INTERFACE I_MotionAxisCommon

PROPERTY AxisState : MC_AxisStates
GET
END_GET
END_PROPERTY

PROPERTY BufferMode : MC_BufferMode
SET
END_SET
END_PROPERTY

PROPERTY Busy : BOOL
GET
END_GET
END_PROPERTY

PROPERTY Cmd : UINT
SET
END_SET
END_PROPERTY

PROPERTY CmdData : UINT
SET
END_SET
END_PROPERTY

PROPERTY CmdHalt : BOOL
GET
END_GET
SET
END_SET
END_PROPERTY

PROPERTY CmdMoveAbsolute : BOOL
GET
END_GET
SET
END_SET
END_PROPERTY

PROPERTY CmdMoveHome : BOOL
GET
END_GET
SET
END_SET
END_PROPERTY

PROPERTY CmdReset : BOOL
GET
END_GET
SET
END_SET
END_PROPERTY

PROPERTY Command : UINT
SET
END_SET
END_PROPERTY

PROPERTY CommandAborted : BOOL
GET
END_GET
END_PROPERTY

PROPERTY CommandData : UINT
SET
END_SET
END_PROPERTY

PROPERTY CommandedHalt : BOOL
GET
END_GET
SET
END_SET
END_PROPERTY

PROPERTY CommandedMoveAbsolute : BOOL
GET
END_GET
SET
END_SET
END_PROPERTY

PROPERTY CommandedReset : BOOL
GET
END_GET
SET
END_SET
END_PROPERTY

PROPERTY Done : BOOL
GET
END_GET
END_PROPERTY

PROPERTY EncoderCount : UDINT
GET
END_GET
END_PROPERTY

PROPERTY Error : BOOL
GET
END_GET
END_PROPERTY

PROPERTY ErrorID : UDINT
GET
END_GET
END_PROPERTY

PROPERTY ErrorMessage : STRING
GET
END_GET
END_PROPERTY

PROPERTY ExecHome : BOOL
GET
END_GET
SET
END_SET
END_PROPERTY

PROPERTY ExecMove : BOOL
GET
END_GET
SET
END_SET
END_PROPERTY

PROPERTY HaltBusy : BOOL
GET
END_GET
END_PROPERTY

PROPERTY HaltDone : BOOL
GET
END_GET
END_PROPERTY

PROPERTY HaltErrorID : UDINT
GET
END_GET
END_PROPERTY

PROPERTY HomeBusy : BOOL
GET
END_GET
END_PROPERTY

PROPERTY HomeDone : BOOL
GET
END_GET
END_PROPERTY

PROPERTY HomeError : BOOL
GET
END_GET
END_PROPERTY

PROPERTY HomeErrorID : UDINT
GET
END_GET
END_PROPERTY

PROPERTY HomeInterrupted : BOOL
GET
END_GET
END_PROPERTY

PROPERTY HomeMode : E_EpicsHomeCmd
GET
END_GET
SET
END_SET
END_PROPERTY

PROPERTY HomePosition : LREAL
GET
END_GET
SET
END_SET
END_PROPERTY

PROPERTY InTargetPosition : BOOL
GET
END_GET
END_PROPERTY

PROPERTY Interrupted : BOOL
GET
END_GET
END_PROPERTY

METHOD InterruptMove
VAR_INPUT
END_VAR
END_METHOD

PROPERTY MeasuredAcceleration : LREAL
GET
END_GET
END_PROPERTY

PROPERTY MeasuredPosition : LREAL
GET
END_GET
END_PROPERTY

PROPERTY MeasuredPositionDiff : LREAL
GET
END_GET
END_PROPERTY

PROPERTY MeasuredVelocity : LREAL
GET
END_GET
END_PROPERTY

PROPERTY ModeOfOperation : SINT
GET
END_GET
SET
END_SET
END_PROPERTY

PROPERTY MoveAbsoluteBusy : BOOL
GET
END_GET
END_PROPERTY

PROPERTY MoveAbsoluteDone : BOOL
GET
END_GET
END_PROPERTY

PROPERTY MoveAbsoluteError : BOOL
GET
END_GET
END_PROPERTY

PROPERTY MoveAbsoluteErrorID : UDINT
GET
END_GET
END_PROPERTY

PROPERTY MoveAbsoluteTargetAcceleration : LREAL
GET
END_GET
SET
END_SET
END_PROPERTY

PROPERTY MoveAbsoluteTargetDeceleration : LREAL
GET
END_GET
SET
END_SET
END_PROPERTY

PROPERTY MoveAbsoluteTargetJerk : LREAL
GET
END_GET
SET
END_SET
END_PROPERTY

PROPERTY MoveAbsoluteTargetPosition : LREAL
GET
END_GET
SET
END_SET
END_PROPERTY

PROPERTY MoveAbsoluteTargetVelocity : LREAL
GET
END_GET
SET
END_SET
END_PROPERTY

PROPERTY MoveMode : E_MoveMode
GET
END_GET
SET
END_SET
END_PROPERTY

PROPERTY Name : STRING
GET
END_GET
SET
END_SET
END_PROPERTY

PROPERTY NCParamsReadInit : BOOL
GET
END_GET
END_PROPERTY

PROPERTY NegativeMotionIsEnabled : BOOL
GET
END_GET
END_PROPERTY

PROPERTY PositiveMotionIsEnabled : BOOL
GET
END_GET
END_PROPERTY

PROPERTY PowerEnable : BOOL
GET
END_GET
SET
END_SET
END_PROPERTY

PROPERTY PowerEnableNegative : BOOL
GET
END_GET
SET
END_SET
END_PROPERTY

PROPERTY PowerEnablePositive : BOOL
GET
END_GET
SET
END_SET
END_PROPERTY

PROPERTY PowerError : BOOL
GET
END_GET
END_PROPERTY

PROPERTY PowerErrorID : UDINT
GET
END_GET
END_PROPERTY

PROPERTY PowerIsEnabled : BOOL
GET
END_GET
END_PROPERTY

PROPERTY PowerOverride : LREAL
GET
END_GET
SET
END_SET
END_PROPERTY

PROPERTY PowerStatus : BOOL
GET
END_GET
END_PROPERTY

PROPERTY RefreshDelay : TIME
GET
END_GET
SET
END_SET
END_PROPERTY

PROPERTY RefVeloSearch : LREAL
GET
END_GET
END_PROPERTY

PROPERTY RefVeloSync : LREAL
GET
END_GET
END_PROPERTY

PROPERTY ResetBusy : BOOL
GET
END_GET
END_PROPERTY

PROPERTY ResetDone : BOOL
GET
END_GET
END_PROPERTY

PROPERTY ResetError : BOOL
GET
END_GET
END_PROPERTY

PROPERTY ResetErrorID : UDINT
GET
END_GET
END_PROPERTY

PROPERTY RestoreDone : BOOL
GET
END_GET
SET
END_SET
END_PROPERTY

PROPERTY RestoreError : BOOL
GET
END_GET
END_PROPERTY

PROPERTY RestoreErrorID : UDINT
GET
END_GET
END_PROPERTY

PROPERTY SavedPosition : LREAL
GET
END_GET
END_PROPERTY

PROPERTY Servo : BOOL
GET
END_GET
SET
END_SET
END_PROPERTY

(* 
	Check all post condition before updating bCommandedMoveAbsolute
	The implmentatation will depend on the axis type
	DS402 NC/Direct axis : Implementation need to check that the drive is in the correct mode before initaiting the move then set bCommandedMoveAbsolute
	MP NC axis : will immediately write to bCommandedMoveAbsolute 
*)
METHOD StartMove : BOOL
VAR_INPUT
END_VAR
END_METHOD

METHOD StopMove
VAR_INPUT
END_VAR
END_METHOD

END_INTERFACE

(* stored: Version 1.1.0.1
   Itf I_MotionAxisCommon: Id {df11a94c-15fb-4aec-9011-b2ef3c6b1fb4}
   Property AxisState: Id {fbced42b-bd0e-4f8b-9d53-090d7101c00b}
   Get Get: Id {3f69a59a-8937-4e06-aeb3-542997f1671d}
   Property BufferMode: Id {38f05b0c-8759-4cb0-852d-594c9ce9b628}
   Set Set: Id {b31efd89-9be0-445c-8e9c-f516f7340490}
   Property Busy: Id {1dc67c19-7944-41b9-ba51-efc9922261f1}
   Get Get: Id {a5860cad-3e89-42b7-8b83-9419c9d09efd}
   Property Cmd: Id {69b39c97-9b90-4d9b-a9e7-485ac83933e1}
   Set Set: Id {abefe843-77e6-4997-be3a-c32a08ca8c8f}
   Property CmdData: Id {054016e0-1db6-4015-9b60-d4eac71effd1}
   Set Set: Id {fc9b83c4-f2f9-46c4-bd97-0ba0143c91d4}
   Property CmdHalt: Id {c0746e6c-e503-4768-b680-1d04f0ae1984}
   Get Get: Id {6a9152b5-e347-4fca-96b2-7284ad169bbc}
   Set Set: Id {98676a7a-0323-4266-9c73-239c40deb92e}
   Property CmdMoveAbsolute: Id {f4037a53-e108-4ca0-9a92-314a66e74287}
   Get Get: Id {447a2d74-14ca-4065-b818-42aaec9a8873}
   Set Set: Id {2137edf8-e503-4512-a064-4f3f78293549}
   Property CmdMoveHome: Id {c447ca24-e237-4885-a9a3-281864c8338b}
   Get Get: Id {bd009231-61d7-4bed-ae68-5c589c9f60c3}
   Set Set: Id {fd07a648-391b-4835-a127-b5f46d9080b8}
   Property CmdReset: Id {d517a452-024b-4976-921a-8fe69a2bf16f}
   Get Get: Id {50257a3a-da8e-4338-964f-dc07fa89e7aa}
   Set Set: Id {056030c6-8ce9-46ea-b6e0-3abbc748c572}
   Property Command: Id {7b9a7e1c-dedf-411f-ad91-f5efd6c329ee}
   Set Set: Id {c20cbc5e-5c11-4ee7-af97-18507def7d36}
   Property CommandAborted: Id {0fa2c2c2-ee04-43d1-b494-0f4602cb897b}
   Get Get: Id {b918462e-6014-4e11-9e53-215e9c34e70a}
   Property CommandData: Id {0e8b4985-8f01-4f1b-8087-81dc02998277}
   Set Set: Id {e5aa3541-32bf-49db-9fad-772fe065c88c}
   Property CommandedHalt: Id {28caa621-b1b5-45c3-948b-355529ae63c2}
   Get Get: Id {9fc451d3-9985-4a65-a079-615be98f9e47}
   Set Set: Id {afbd26a2-5d4f-4673-a5ff-92792f920642}
   Property CommandedMoveAbsolute: Id {be1022ab-c175-45cf-b747-4904f7dbb61a}
   Get Get: Id {2b465d88-c80e-452d-bd64-a4daa37a937f}
   Set Set: Id {148eb03e-69c6-4884-b363-b91c6e29515e}
   Property CommandedReset: Id {cd7e8bfd-a0cf-4671-a69b-1557a160bd00}
   Get Get: Id {cc6afb54-414e-4354-b571-2acc42bfca27}
   Set Set: Id {367e203b-5f9b-41d7-9061-a806fa5317d7}
   Property Done: Id {7ff11c7c-614b-47cb-baec-d0e1b99b56ef}
   Get Get: Id {731f59b1-4ebc-46a2-8ec3-b8482a33696e}
   Property EncoderCount: Id {9e7da4f2-c20f-41ff-89bb-b6a6d51aa2c8}
   Get Get: Id {e6419d2f-35cd-4088-84a8-5db9b615087b}
   Property Error: Id {1839383d-e5fd-4221-a255-d379f863c6e8}
   Get Get: Id {3b6a6767-2e6d-4d83-ac0a-858e93b4acb4}
   Property ErrorID: Id {a8ca6773-3b68-40ff-aa9d-b90cfd491bbf}
   Get Get: Id {3c8f7f0c-cdf8-46a2-b2ed-eae80213300d}
   Property ErrorMessage: Id {62e7f2d7-0787-4e90-bcb4-6a79cccb37fe}
   Get Get: Id {540b8f36-640c-487f-bfb4-5e6df636128d}
   Property ExecHome: Id {6e6bf230-720c-4613-80af-c8c009118fd1}
   Get Get: Id {6125f9cc-b415-4a4e-b052-4c188af3488f}
   Set Set: Id {7f9e6770-dd66-4322-8ad8-27eaa7f2abde}
   Property ExecMove: Id {9fe3d498-d752-48dc-aa3d-5d4c1306ffed}
   Get Get: Id {a97d3154-60d9-4bed-b64b-6f7f0fa20999}
   Set Set: Id {df2886f7-a831-4b24-b707-10da4aeec211}
   Property HaltBusy: Id {5eefa523-d59e-4ef7-b5af-021b09543db4}
   Get Get: Id {e59b7e42-9140-4829-bc23-b10577952d4c}
   Property HaltDone: Id {2708b684-0763-4c58-ad74-2f54f4c3351c}
   Get Get: Id {1696e0d8-0e21-4edb-aa6d-6c70bfdba3fc}
   Property HaltErrorID: Id {76c342d8-ef7a-4cbf-b33e-fe9701803b90}
   Get Get: Id {84f9ea8e-6e1e-480a-86db-80a8046724f4}
   Property HomeBusy: Id {d6d79540-89df-4e37-8d40-761027f4650a}
   Get Get: Id {2085b480-133e-431e-af2b-2e28067f5fcf}
   Property HomeDone: Id {6d82612d-3be0-411d-9fbb-4db9d5b30e7a}
   Get Get: Id {dc264365-5ed4-4cc8-8938-a641a37a624b}
   Property HomeError: Id {66345dd5-8f9b-4c6e-862e-018015cab45f}
   Get Get: Id {bf4a9cda-c749-44e3-b222-0aa2dcfcebdb}
   Property HomeErrorID: Id {5637a821-11d4-4cf6-b60b-88d54de78092}
   Get Get: Id {522d3d81-d3e7-4960-90e6-f89bf9e2f7eb}
   Property HomeInterrupted: Id {e35df6e5-941d-4778-a7be-e76d3f381d59}
   Get Get: Id {58767f79-ed58-4276-8041-a41052c97a6b}
   Property HomeMode: Id {32879e99-b015-407a-b611-ffd5ee8ac39d}
   Get Get: Id {16a9aefe-77f3-400a-84d1-c01ba499762b}
   Set Set: Id {7d19f097-4494-4927-be4b-078feb862d60}
   Property HomePosition: Id {292c1204-dc74-485b-8911-177c01a78ff8}
   Get Get: Id {9ffd7eeb-12d8-4c9d-8056-57cabd96be13}
   Set Set: Id {3692be77-4178-4aa1-b1e2-16325bc48cb0}
   Property InTargetPosition: Id {79a34037-a39e-4bee-ab9e-d3c72c400a3c}
   Get Get: Id {c1b81aa3-9460-4489-85a7-c42e28336f83}
   Property Interrupted: Id {498fa652-b5b3-4e1f-976d-8ce99932c93a}
   Get Get: Id {2c6824d4-b3f4-460d-9f3f-bc04fc1c06c7}
   Method InterruptMove: Id {303223bb-9993-4d05-b3de-df5e0ce6e8a3}
   Property MeasuredAcceleration: Id {d4d9e574-a194-4fa2-98b9-07d056a1260a}
   Get Get: Id {64393f7d-024e-4f33-8143-f1be9ffe5b8f}
   Property MeasuredPosition: Id {d63c1cdc-d7a8-436e-8781-271d2fcb7da2}
   Get Get: Id {36e1d037-35d3-410b-bb6f-e4f6e0d800dc}
   Property MeasuredPositionDiff: Id {4962ee10-def8-4f9d-bf3b-0b44ac0ece59}
   Get Get: Id {fc230d1f-c943-4ec1-a46d-a7979d2b7069}
   Property MeasuredVelocity: Id {ba169ffc-f0a6-4913-8469-66deff516709}
   Get Get: Id {62daf172-9d22-4bb4-bfac-abdfd22e6c7b}
   Property ModeOfOperation: Id {e6ef5f87-d9f5-4819-a545-2bdc671caace}
   Get Get: Id {5767ff6c-d328-42fc-a0a0-bd49b1295ca0}
   Set Set: Id {c3f1cd01-5c5f-4eb4-afce-893c68097624}
   Property MoveAbsoluteBusy: Id {f8fb30ef-d277-418f-982b-66ef86e1769d}
   Get Get: Id {11b339b5-cdec-49fb-9600-a6ec69bc6a16}
   Property MoveAbsoluteDone: Id {84978858-3bb9-4917-be38-de8a68ac208b}
   Get Get: Id {129da105-f372-4faf-add9-30e139e5f062}
   Property MoveAbsoluteError: Id {64cf4975-3274-4a57-9bc5-8610f16695ba}
   Get Get: Id {681cadf4-083a-4ae4-a53c-86cf46221723}
   Property MoveAbsoluteErrorID: Id {4fb23927-b236-4114-ae37-f615a1b8edc0}
   Get Get: Id {a023c07f-7952-4ec4-83ec-1efda5ff2614}
   Property MoveAbsoluteTargetAcceleration: Id {70a35961-bee7-4b46-b0a3-6d71eaea287d}
   Get Get: Id {9898cff6-ce1f-4fb8-8f53-4ba3d7d4fea1}
   Set Set: Id {b2459bb9-7080-49b9-ae3a-a918cd839621}
   Property MoveAbsoluteTargetDeceleration: Id {31845d61-2b46-4eb7-89e1-f67edbd56c4f}
   Get Get: Id {9a64bf3b-7a3b-4dec-a769-9b31e5a86434}
   Set Set: Id {e7ada26d-8451-438f-b463-e10f2d3a1bb8}
   Property MoveAbsoluteTargetJerk: Id {9119fca5-a884-4a17-a499-ebd775946ce3}
   Get Get: Id {1a98813c-01e8-4cb0-8272-d799fe855c2f}
   Set Set: Id {fcaf00f7-169a-4518-82c4-db7d885f20c5}
   Property MoveAbsoluteTargetPosition: Id {4c3ad4b2-e392-4b88-8a83-082f941a6830}
   Get Get: Id {8a09bba2-a387-469e-8361-0e2306956cba}
   Set Set: Id {c58fc251-226c-4365-badb-dca9ec823ab7}
   Property MoveAbsoluteTargetVelocity: Id {08e71f81-65e6-4cad-a488-7ef932c2b524}
   Get Get: Id {d4d23ccf-3369-4604-993d-56d3faa062bc}
   Set Set: Id {0be80c1e-730f-40bc-8e47-969d994de88e}
   Property MoveMode: Id {05f924a5-d3a6-4da7-ab50-fcad0580fbfb}
   Get Get: Id {4e619b19-1227-4aa9-97bd-f7e260dcc6cd}
   Set Set: Id {2987c28d-902f-4e1a-bce2-2b0a7c7390d5}
   Property Name: Id {0c6fd7a6-29c0-4c88-879f-f0f43862e70a}
   Get Get: Id {0df1c16f-fce7-44ce-a865-4fda8703479c}
   Set Set: Id {50a58ed7-b3ae-45d2-8b55-54fab7befe10}
   Property NCParamsReadInit: Id {f843168c-ca4c-4733-b6db-f83934f20ac1}
   Get Get: Id {9c60541a-3e75-4e37-92d5-dc139cd07934}
   Property NegativeMotionIsEnabled: Id {89f73a4c-6b65-4069-892b-fbfc7e7d2963}
   Get Get: Id {82333464-dc32-4ef8-bfed-612699606e4b}
   Property PositiveMotionIsEnabled: Id {52b21291-5115-4fe8-b5cd-5d002408c68b}
   Get Get: Id {1b2b33a3-a699-41d1-89bf-9eec4d0a49ca}
   Property PowerEnable: Id {8f4626d6-0f8b-4b9d-a413-29dca15842e6}
   Get Get: Id {80cde4e4-17e9-4a07-a9cc-6347ce732266}
   Set Set: Id {b3427a42-2fec-45a1-86c8-2c735642631f}
   Property PowerEnableNegative: Id {a552419c-1e47-4ba6-86f3-9cd43b6c7d4f}
   Get Get: Id {c8e9c776-921f-42c7-a895-e64aa928906d}
   Set Set: Id {2d84af61-aa81-442f-87dd-3dcea000019a}
   Property PowerEnablePositive: Id {8a310391-dab0-4dd4-84ea-7e42d91a1c1b}
   Get Get: Id {9f36b795-1fb8-4212-83b1-d67198dca149}
   Set Set: Id {ba7d2aa7-0ae3-4c74-874c-2d6ae8f7c7cf}
   Property PowerError: Id {cb1b5b40-b70d-4a67-958a-9b06cfba612b}
   Get Get: Id {ae2b0ff5-5ffb-44e3-b875-297aa814c673}
   Property PowerErrorID: Id {4aee72fa-f2a7-431e-b4b4-0b9354d8eb3f}
   Get Get: Id {a54d7cf3-a137-4078-938e-e669e7c312e2}
   Property PowerIsEnabled: Id {1be1dbac-9180-4e18-8d7d-7ac4fb3a523a}
   Get Get: Id {dae81c77-289b-440a-8b61-e8ef6a37bede}
   Property PowerOverride: Id {db8164ef-c0bf-4e70-a366-22ab4e209738}
   Get Get: Id {a17504c2-efbb-4971-b4f3-eedbd364db39}
   Set Set: Id {ff31e593-5cb0-4acb-982d-4ad437bb4265}
   Property PowerStatus: Id {ec6d63e1-de25-46f8-a4c8-a861493a5d55}
   Get Get: Id {5341a077-011d-4b04-9806-ab379cb1f954}
   Property RefreshDelay: Id {9a60c61b-0084-4420-be8f-035904aea924}
   Get Get: Id {f1806e9b-0dce-4abd-af1d-83272cb8df1e}
   Set Set: Id {24faa0ad-b9ca-4984-a659-ab17c9d097d8}
   Property RefVeloSearch: Id {06c09a70-377d-482c-a85b-e4912b1ba011}
   Get Get: Id {1e34b3e3-2a6f-40c7-b27b-eeacf2ee48da}
   Property RefVeloSync: Id {ad7860fb-e8a6-42b6-aaff-223373b4f98f}
   Get Get: Id {62cd0a9d-dc15-48af-ae9d-14d810b2fe9f}
   Property ResetBusy: Id {252e8874-c509-40df-a935-8a5f3cbe2b7a}
   Get Get: Id {1352f413-28b0-47c7-89f3-68206fd5c6bb}
   Property ResetDone: Id {d4e08fc6-eeda-4353-a1d6-7047dbfb6a8a}
   Get Get: Id {754bf460-2d23-4adc-8924-46cc6786b79b}
   Property ResetError: Id {492c4d78-fea4-491d-9af5-1a5800d3ff0f}
   Get Get: Id {9f4ff4de-0fc6-450d-a532-1e53e644e0fc}
   Property ResetErrorID: Id {7ec9a9da-2ba3-442e-8c3f-a80607933d95}
   Get Get: Id {0adcb703-0fab-4a7a-94a7-18c9597f870e}
   Property RestoreDone: Id {852d5da2-20f3-40a4-8ab0-8b0ebb2ca285}
   Get Get: Id {4f3b62f8-9947-4e8d-a9cf-f23f4d32cb01}
   Set Set: Id {11f68748-f280-450f-b307-949684cb9a43}
   Property RestoreError: Id {80815cd7-c76d-4675-bb97-e801d3dcea69}
   Get Get: Id {dbe76bd4-2085-47ed-82a9-7ce3e56236f5}
   Property RestoreErrorID: Id {14478e39-3848-4591-86df-eb5530d2d0db}
   Get Get: Id {369bf874-f43c-4d30-9d9f-b15735e7d325}
   Property SavedPosition: Id {c75abb61-130a-473f-af2a-684df4a5b1a1}
   Get Get: Id {9c9bf27a-4d43-4c82-8ef0-db2f0c4f18cb}
   Property Servo: Id {1e11ef79-2846-41f4-a9ea-4e652e593f38}
   Get Get: Id {ac50adb8-becc-4f8c-9005-b9e3971381d2}
   Set Set: Id {2ae0d9a9-000d-4e26-8a6d-320c30eb8752}
   Method StartMove: Id {d1e01015-af1a-4437-ac2e-693a8f3c4a64}
   Method StopMove: Id {2531f2ec-0334-47a8-bd79-645624a1e210} *)
